(* IEC 61131-3 sources: s22-soft-shell/st_interpret/tests/test_inputs/execution/st_stretch, 1 file *)

(* ---- stretch_pow.st ---- *)
PROGRAM stretch_pow
VAR
    a: int;
    ST_TESTING_RESULT : bool;
END_VAR
    a := 3 ** 3;
        ST_TESTING_RESULT := (a = 27);
END_PROGRAM
